FUNCTION_BLOCK FB_AdjustmentProcess
VAR_INPUT
    bEnable          : BOOL;
    bAbort           : BOOL;
    bStopRequest     : BOOL;
    bMachinePrepared : BOOL;
    bStartRequest    : BOOL;
    bDoneAck         : BOOL;

    // 与Screwdriver流程之间的保持型业务握手。
    bSecondTightenDone : BOOL;
    bReworkLoosenDone  : BOOL;

    // 保留原输入符号以兼容现有监控；协调器给它与二次拧紧Done相同的值。
    bRetractPermit : BOOL;
END_VAR

VAR_IN_OUT
    ioAdjustGripperAction : FB_GripperAction;
    ioAdjustGripper       : ST_GripperInterface;
    stAxisX               : ST_AxisInterface;
    stAxisY               : ST_AxisInterface;
    stAxisZ               : ST_AxisInterface;
END_VAR

VAR_OUTPUT
    bAdjustmentReady   : BOOL; // 兼容诊断：与二次拧紧请求保持一致
    bAdjustmentDone    : BOOL;
    bAdjustmentBusy    : BOOL;
    bAdjustmentQualified : BOOL;
	bAdjustmentOutOfRange : BOOL;
    bRequestSecondTighten : BOOL;
    bRequestReworkLoosen  : BOOL;// 当前件超出Adjustment可调整范围。
    bVisionTimeout     : BOOL;
    bVisionFault       : BOOL;
    bFallbackUsed      : BOOL;
    eVisionError       : E_VisionError := E_VisionError.None;
    fVisionCoaxiality  : LREAL;
    fCorrectionX       : LREAL;
    fCorrectionY       : LREAL;
    nAdjustCount       : UINT;
    nReworkCount       : UINT;
    bError             : BOOL;
    bGripperError      : BOOL;
    uiErrorAxis        : UINT;
    udErrorCode        : UDINT;
    eStep              : E_AdjustmentStep := E_AdjustmentStep.Idle;
    bAdjustGripperActionExecute : BOOL;
    eAdjustGripperActionCommand : E_GripperCommand := E_GripperCommand.None;
END_VAR

VAR
    fXWork : LREAL;
    fYWork : LREAL;
    fZWork : LREAL;
    fXStandby : LREAL;
    fYStandby : LREAL;
    fZSafe : LREAL;
    fXVelocity : LREAL;
    fYVelocity : LREAL;
    fZVelocity : LREAL;
    fPositionTolerance : LREAL;
    tMoveTimeout : TIME;

	//==============================================================
	// Adjustment最终被PLC接受并真正下发给轴的绝对目标
	//==============================================================
	fAdjustTargetX : LREAL;
	fAdjustTargetY : LREAL;
	
	
	//==============================================================
	// 本次Coax修正计算出的候选绝对目标
	//
	// Candidate = 当前实际位置 + Python修正量
	//
	// 候选值只有通过±最大修正范围检查后，
	// 才允许写入fAdjustTargetX/Y。
	//==============================================================
	fCandidateTargetX : LREAL;
	fCandidateTargetY : LREAL;
	
	
	//==============================================================
	// 修正目标范围诊断
	//==============================================================
	bCorrectionXOutOfRange : BOOL;
	bCorrectionYOutOfRange : BOOL;
	
	
	bVisionWithinTolerance : BOOL;
	
    fbMoveTimeout : TON;
    fbCoaxVision : FB_CoaxVision;
    // 当前逻辑检测点的额外检测计数；Retry路径不得清零。
    nCoaxRetryCount : UINT;
    fbCoaxRetryDelay : TON;
    bTimerRestart : BOOL;
    eTimedStep : E_AdjustmentStep := E_AdjustmentStep.Idle;
    bTimedMovement : BOOL;
    uiMovingAxis : UINT;

    bXIssued : BOOL;
    bYIssued : BOOL;
    bZIssued : BOOL;
    bXDone : BOOL;
    bYDone : BOOL;
    bZDone : BOOL;
END_VAR

// 沿用现有PositionConfig和MotionConfig；视觉工艺、次数和超时分别来自
// ProcessConfig与CommunicationConfig，FB内部不保存第二套参数源。
fXWork := GVL_PositionConfig.stAdjustment.stWork.X;
fYWork := GVL_PositionConfig.stAdjustment.stWork.Y;
fZWork := GVL_PositionConfig.stAdjustment.stWork.Z;
fXStandby := GVL_PositionConfig.stAdjustment.stReady.X;
fYStandby := GVL_PositionConfig.stAdjustment.stReady.Y;
fZSafe := GVL_PositionConfig.stAdjustment.stReady.Z;
fXVelocity := GVL_MotionConfig.stAdjustment.stX.fVelocity;
fYVelocity := GVL_MotionConfig.stAdjustment.stY.fVelocity;
fZVelocity := GVL_MotionConfig.stAdjustment.stZ.fVelocity;
fPositionTolerance := GVL_MotionConfig.stAdjustment.fPositionTolerance;
tMoveTimeout := GVL_MotionConfig.stAdjustment.tMoveTimeout;

bTimerRestart := (eStep <> eTimedStep);
eTimedStep := eStep;
bTimedMovement :=
    (eStep = E_AdjustmentStep.MoveXYToWork)
    OR (eStep = E_AdjustmentStep.LowerZToWork)
    OR (eStep = E_AdjustmentStep.WaitCorrectionXY)
    OR (eStep = E_AdjustmentStep.LiftZToSafe)
    OR (eStep = E_AdjustmentStep.ReturnXYToStandby);

IF bTimedMovement THEN
    CASE eStep OF
        E_AdjustmentStep.LowerZToWork,
        E_AdjustmentStep.LiftZToSafe:
            uiMovingAxis := GVL_AxisIndex.AdjustmentZ;

        E_AdjustmentStep.MoveXYToWork,
        E_AdjustmentStep.WaitCorrectionXY,
        E_AdjustmentStep.ReturnXYToStandby:
            IF NOT bXDone THEN
                uiMovingAxis := GVL_AxisIndex.AdjustmentX;
            ELSE
                uiMovingAxis := GVL_AxisIndex.AdjustmentY;
            END_IF;
    END_CASE;
END_IF;

fbMoveTimeout(
    IN := bEnable AND NOT bAbort AND bTimedMovement AND NOT bTimerRestart,
    PT := tMoveTimeout
);

stAxisX.AutoCmd.bMoveAbs := FALSE;
stAxisY.AutoCmd.bMoveAbs := FALSE;
stAxisZ.AutoCmd.bMoveAbs := FALSE;
bAdjustGripperActionExecute := FALSE;
eAdjustGripperActionCommand := E_GripperCommand.None;

// Retry属于Adjustment工艺层；两个Delay状态均撤销视觉bExecute。
// 每扫描只调用一次TON，离开Delay状态或停止/取消时复位。
fbCoaxRetryDelay(
    IN := bEnable AND NOT bAbort AND NOT bStopRequest
          AND ((eStep = E_AdjustmentStep.WaitMeasureRetryDelay)
               OR (eStep = E_AdjustmentStep.WaitFinalMeasureRetryDelay)),
    PT := GVL_ProcessConfig.stAdjustment.tCoaxRetryDelay
);

// Process只保持执行请求并消费强类型结果；ADS、RequestId、ResultId和Timeout
// 全部封装在FB_CoaxVision -> FB_VisionRequest中。
fbCoaxVision(
    bExecute := bEnable
                AND NOT bAbort
                AND
                (
                    (eStep = E_AdjustmentStep.WaitMeasureResult)
                    OR (eStep = E_AdjustmentStep.WaitFinalMeasure)
                ),
    bCancel := bStopRequest OR bAbort
);

IF NOT bEnable OR bAbort THEN
    IF bMachinePrepared THEN
        ioAdjustGripperAction(
            bExecute := FALSE,
            eCommand := E_GripperCommand.None,
            bCancel := bStopRequest OR bAbort,
            tAcceptTimeout := GVL_ProcessConfig.stGripper.tAcceptTimeout,
            tResultTimeout := GVL_ProcessConfig.stGripper.tResultTimeout,
            ioGripper := ioAdjustGripper
        );
    END_IF;

    bAdjustmentReady := FALSE;
    bAdjustmentDone := FALSE;
    bAdjustmentBusy := FALSE;
    bAdjustmentQualified := FALSE;
	bAdjustmentOutOfRange := FALSE;
    bRequestSecondTighten := FALSE;
    bRequestReworkLoosen := FALSE;
    bVisionTimeout := FALSE;
    bVisionFault := FALSE;
    bFallbackUsed := FALSE;
    eVisionError := E_VisionError.None;
    fCorrectionX := 0.0;
    fCorrectionY := 0.0;
	fCandidateTargetX := 0.0;
	fCandidateTargetY := 0.0;
	bCorrectionXOutOfRange := FALSE;
	bCorrectionYOutOfRange := FALSE;
    nAdjustCount := 0;
    nReworkCount := 0;
    nCoaxRetryCount := 0;
    bError := FALSE;
    bGripperError := FALSE;
    uiErrorAxis := 0;
    udErrorCode := TO_UDINT(E_ScrewdriverErrorCode.None);
    bXIssued := FALSE;
    bYIssued := FALSE;
    bZIssued := FALSE;
    bXDone := FALSE;
    bYDone := FALSE;
    bZDone := FALSE;
    eStep := E_AdjustmentStep.Idle;
    RETURN;
END_IF;

IF (eStep = E_AdjustmentStep.Idle) AND bStartRequest THEN

 	//==========================================================
    // 新工件开始，清除上一件质量结果。
    //==========================================================
    bAdjustmentQualified := FALSE;
	bAdjustmentOutOfRange := FALSE;

    bVisionTimeout := FALSE;
    bVisionFault := FALSE;
    bFallbackUsed := FALSE;
    eVisionError := E_VisionError.None;

    bVisionWithinTolerance := FALSE;

    fVisionCoaxiality := 0.0;

    fCorrectionX := 0.0;
    fCorrectionY := 0.0;

    // 初始接受目标仍然从Adjustment工作位置开始。
    fAdjustTargetX := fXWork;
    fAdjustTargetY := fYWork;

    // 候选目标初始化到工作位置。
    fCandidateTargetX := fXWork;
    fCandidateTargetY := fYWork;

    // 清除上一件产品的范围诊断。
    bCorrectionXOutOfRange := FALSE;
    bCorrectionYOutOfRange := FALSE;

    nAdjustCount := 0;
    nReworkCount := 0;
    nCoaxRetryCount := 0;

    bXIssued := FALSE;
    bYIssued := FALSE;
    bXDone := FALSE;
    bYDone := FALSE;

    eStep := E_AdjustmentStep.MoveXYToWork;
END_IF;

// 准备阶段结束后，COM4命令权归本FB；Open持续到最终质量结果确定。
IF bMachinePrepared THEN
    IF eStep = E_AdjustmentStep.OpenGripper THEN
        bAdjustGripperActionExecute := TRUE;
        eAdjustGripperActionCommand := E_GripperCommand.Open;
    ELSIF eStep = E_AdjustmentStep.CloseGripper THEN
        bAdjustGripperActionExecute := TRUE;
        eAdjustGripperActionCommand := E_GripperCommand.Close;
    END_IF;

    ioAdjustGripperAction(
        bExecute := bAdjustGripperActionExecute,
        eCommand := eAdjustGripperActionCommand,
        bCancel := bStopRequest OR bAbort,
        tAcceptTimeout := GVL_ProcessConfig.stGripper.tAcceptTimeout,
        tResultTimeout := GVL_ProcessConfig.stGripper.tResultTimeout,
        ioGripper := ioAdjustGripper
    );
END_IF;

IF stAxisX.Alarm.bError OR stAxisY.Alarm.bError OR stAxisZ.Alarm.bError THEN
    bError := TRUE;
    bGripperError := FALSE;
    eStep := E_AdjustmentStep.Error;
    IF stAxisX.Alarm.bError THEN
        uiErrorAxis := GVL_AxisIndex.AdjustmentX;
        udErrorCode := stAxisX.Alarm.nErrorID;
    ELSIF stAxisY.Alarm.bError THEN
        uiErrorAxis := GVL_AxisIndex.AdjustmentY;
        udErrorCode := stAxisY.Alarm.nErrorID;
    ELSE
        uiErrorAxis := GVL_AxisIndex.AdjustmentZ;
        udErrorCode := stAxisZ.Alarm.nErrorID;
    END_IF;
END_IF;

IF ioAdjustGripperAction.bError
    AND ((eStep = E_AdjustmentStep.OpenGripper)
         OR (eStep = E_AdjustmentStep.CloseGripper))
THEN
    bError := TRUE;
    bGripperError := TRUE;
    uiErrorAxis := 0;
    IF ioAdjustGripperAction.udErrorCode <> 0 THEN
        udErrorCode := ioAdjustGripperAction.udErrorCode;
    ELSE
        udErrorCode := TO_UDINT(E_ScrewdriverErrorCode.AdjustmentGripperFailed);
    END_IF;
    eStep := E_AdjustmentStep.Error;
END_IF;

IF fbMoveTimeout.Q AND NOT bError THEN
    bError := TRUE;
    bGripperError := FALSE;
    uiErrorAxis := uiMovingAxis;
    udErrorCode := TO_UDINT(E_ScrewdriverErrorCode.PositionTimeout);
    eStep := E_AdjustmentStep.Error;
END_IF;

CASE eStep OF
    E_AdjustmentStep.Idle:
        bAdjustmentDone := FALSE;

    E_AdjustmentStep.MoveXYToWork:
        IF NOT bXDone THEN
            bXDone := M_MoveAxisAbsolute(fTarget := fXWork, fVelocity := fXVelocity,
                uiAxis := GVL_AxisIndex.AdjustmentX, ioIssued := bXIssued, ioAxis := stAxisX);
        END_IF;
        IF NOT bYDone THEN
            bYDone := M_MoveAxisAbsolute(fTarget := fYWork, fVelocity := fYVelocity,
                uiAxis := GVL_AxisIndex.AdjustmentY, ioIssued := bYIssued, ioAxis := stAxisY);
        END_IF;
        IF bXDone AND bYDone THEN
            fAdjustTargetX := fXWork;
            fAdjustTargetY := fYWork;
            bZIssued := FALSE;
            bZDone := FALSE;
            eStep := E_AdjustmentStep.LowerZToWork;
        END_IF;

    E_AdjustmentStep.LowerZToWork:
        bZDone := M_MoveAxisAbsolute(fTarget := fZWork, fVelocity := fZVelocity,
            uiAxis := GVL_AxisIndex.AdjustmentZ, ioIssued := bZIssued, ioAxis := stAxisZ);
        IF bZDone THEN
            eStep := E_AdjustmentStep.OpenGripper;
        END_IF;

    E_AdjustmentStep.OpenGripper:
        IF ioAdjustGripperAction.bDone THEN
            eStep := E_AdjustmentStep.PrepareMeasurement;
        END_IF;

    E_AdjustmentStep.PrepareMeasurement:
        // 工作位的首次逻辑检测点。Retry直接回RequestMeasure，不经过这里。
        nCoaxRetryCount := 0;
        fCorrectionX := 0.0;
        fCorrectionY := 0.0;
        bVisionWithinTolerance := FALSE;
        // Simulation与Camera都从FB_CoaxVision的统一结果出口获取数据。
        eStep := E_AdjustmentStep.RequestMeasure;

    E_AdjustmentStep.RequestMeasure:
        fCorrectionX := 0.0;
        fCorrectionY := 0.0;
        bVisionWithinTolerance := FALSE;
        eStep := E_AdjustmentStep.WaitMeasureResult;

    E_AdjustmentStep.WaitMeasureResult:
        // Cancelled/Stop由现有Stop/Abort/Reset体系清理，不消费为产品结果。
        IF fbCoaxVision.bDone
            AND NOT bStopRequest
            AND (fbCoaxVision.eVisionError <> E_VisionError.Cancelled)
        THEN
            IF fbCoaxVision.bVisionFault THEN
                IF ((fbCoaxVision.eVisionError = E_VisionError.InvalidResult)
                    OR (fbCoaxVision.eVisionError = E_VisionError.Timeout))
                    AND (nCoaxRetryCount < GVL_ProcessConfig.stAdjustment.nCoaxMaxRetryCount)
                THEN
                    // 暂时失败不锁存工件级诊断；下一次执行创建新的RequestId。
                    nCoaxRetryCount := nCoaxRetryCount + 1;
                    eStep := E_AdjustmentStep.WaitMeasureRetryDelay;
                ELSE
                    // Retry耗尽，或Offline/ServiceFault：当前件不合格，正常撤离。
                    bVisionFault := TRUE;
                    bFallbackUsed := fbCoaxVision.bFallbackUsed;
                    eVisionError := fbCoaxVision.eVisionError;
                    bVisionTimeout :=
                        fbCoaxVision.eVisionError = E_VisionError.Timeout;
                    bAdjustmentQualified := FALSE;
                    eStep := E_AdjustmentStep.CloseGripper;
                END_IF;
            ELSE
                // 仅有效测量进入工艺判断；恢复成功不保留中间失败诊断。
                bVisionFault := FALSE;
                bVisionTimeout := FALSE;
                bFallbackUsed := FALSE;
                eVisionError := E_VisionError.None;
                fVisionCoaxiality := fbCoaxVision.stResult.fCoaxiality;
                fCorrectionX := fbCoaxVision.stResult.fCorrectionX;
                fCorrectionY := fbCoaxVision.stResult.fCorrectionY;
                bVisionWithinTolerance :=
                    fVisionCoaxiality <= GVL_ProcessConfig.stAdjustment.fAdjustTolerance;
                eStep := E_AdjustmentStep.EvaluateAdjustment;
            END_IF;
        END_IF;

    E_AdjustmentStep.WaitMeasureRetryDelay:
        // 本扫描fbCoaxVision.bExecute=FALSE，PT=0时也先正常复位旧事务。
        IF fbCoaxRetryDelay.Q AND NOT bStopRequest THEN
            // 同一逻辑检测点的Retry，保留nCoaxRetryCount。
            eStep := E_AdjustmentStep.RequestMeasure;
        END_IF;

    E_AdjustmentStep.EvaluateAdjustment:

		//==========================================================
		// 情况1：
		// 当前同轴度已经达到调整容差；
		//
		// 或者：
		// 已经达到本轮最大允许调整次数。
		//
		// 此时不再进行新的AdjustmentXY修正。
		//==========================================================
		IF
			bVisionWithinTolerance
			OR
			(
				nAdjustCount
				>= GVL_ProcessConfig.stAdjustment.nMaxAdjustCount
			)
		THEN
	
			eStep :=
				E_AdjustmentStep.RequestSecondTighten;
	
	
		ELSE
	
			//======================================================
			// 统一视觉结果中的Correction为机械相对修正位移，单位mm。
			// Camera映射与比例标定由Python完成；Simulation由FB_CoaxVision生成。
			// 本流程直接消费Correction，不再根据Delta映射或换算。
			// Candidate = ActualPosition + Correction
			//======================================================	
			fCandidateTargetX :=
				stAxisX.Data.fActPosition
				+ fCorrectionX;
	
			fCandidateTargetY :=
				stAxisY.Data.fActPosition
				+ fCorrectionY;
	
	
			//======================================================
			// 检查候选位置是否仍然处于
			//
			// Adjustment工作位置 ± 最大允许调整范围
			//
			// 这里检查的是累计机械偏移，
			// 而不是单次Delta大小。
			//======================================================
	
			bCorrectionXOutOfRange :=
				ABS(
					fCandidateTargetX
					- fXWork
				)
				>
				GVL_ProcessConfig.stAdjustment.fMaxCorrectionX;
	
			bCorrectionYOutOfRange :=
				ABS(
					fCandidateTargetY
					- fYWork
				)
				>
				GVL_ProcessConfig.stAdjustment.fMaxCorrectionY;
	
	
			//======================================================
			// 任意一个方向越界：
			//
			// X/Y作为同一次二维Coax修正，
			// 不允许只执行其中一根轴。
			//
			// 所以两根轴都不运动。
			//======================================================
			IF
				bCorrectionXOutOfRange
				OR
				bCorrectionYOutOfRange
			THEN
			
				// 超范围仅是调整能力诊断；不接受Candidate，不移动任意一根轴。
				// 仍执行二次拧紧，最终质量仅由Final Coax决定。
				bAdjustmentOutOfRange := TRUE;
				bXIssued := FALSE;
				bYIssued := FALSE;
				bXDone := FALSE;
				bYDone := FALSE;
				eStep := E_AdjustmentStep.RequestSecondTighten;

			ELSE
			
				//==========================================================
				// X/Y候选目标均处于允许Adjustment修正窗口内。
				// 正式接受Candidate作为新的轴绝对目标。
				//==========================================================
			
				bAdjustmentOutOfRange := FALSE;
			
				fAdjustTargetX :=
					fCandidateTargetX;
			
				fAdjustTargetY :=
					fCandidateTargetY;
			
				nAdjustCount :=
					nAdjustCount + 1;
			
				eStep :=
					E_AdjustmentStep.StartCorrectionXY;
			
			END_IF;

		END_IF;

    E_AdjustmentStep.StartCorrectionXY:
        bXIssued := FALSE;
        bYIssued := FALSE;
        bXDone := FALSE;
        bYDone := FALSE;
        eStep := E_AdjustmentStep.WaitCorrectionXY;

    E_AdjustmentStep.WaitCorrectionXY:
        // Z保持工作高度，X/Y同时向通过工艺范围检查后的绝对目标运动。
        IF NOT bXDone THEN
            bXDone := M_MoveAxisAbsolute(fTarget := fAdjustTargetX, fVelocity := fXVelocity,
                uiAxis := GVL_AxisIndex.AdjustmentX, ioIssued := bXIssued, ioAxis := stAxisX);
        END_IF;
        IF NOT bYDone THEN
            bYDone := M_MoveAxisAbsolute(fTarget := fAdjustTargetY, fVelocity := fYVelocity,
                uiAxis := GVL_AxisIndex.AdjustmentY, ioIssued := bYIssued, ioAxis := stAxisY);
        END_IF;
        IF bXDone AND bYDone THEN
            // 每次XY修正完成后开始新的逻辑检测点。
            nCoaxRetryCount := 0;
            eStep := E_AdjustmentStep.RequestMeasure;
        END_IF;

    E_AdjustmentStep.RequestSecondTighten:
        eStep := E_AdjustmentStep.WaitSecondTighten;

    E_AdjustmentStep.WaitSecondTighten:
        IF bSecondTightenDone OR bRetractPermit THEN
            // 二次拧紧已完成；Final是独立的逻辑检测点。
            nCoaxRetryCount := 0;
            eStep := E_AdjustmentStep.RequestFinalMeasure;
        END_IF;

    E_AdjustmentStep.RequestFinalMeasure:
        fCorrectionX := 0.0;
        fCorrectionY := 0.0;
        bVisionWithinTolerance := FALSE;
        eStep := E_AdjustmentStep.WaitFinalMeasure;

    E_AdjustmentStep.WaitFinalMeasure:
        // Cancelled/Stop由现有Stop/Abort/Reset体系清理，不消费为产品结果。
        IF fbCoaxVision.bDone
            AND NOT bStopRequest
            AND (fbCoaxVision.eVisionError <> E_VisionError.Cancelled)
        THEN
            IF fbCoaxVision.bVisionFault THEN
                IF ((fbCoaxVision.eVisionError = E_VisionError.InvalidResult)
                    OR (fbCoaxVision.eVisionError = E_VisionError.Timeout))
                    AND (nCoaxRetryCount < GVL_ProcessConfig.stAdjustment.nCoaxMaxRetryCount)
                THEN
                    // 暂时失败不锁存工件级诊断；下一次执行创建新的RequestId。
                    nCoaxRetryCount := nCoaxRetryCount + 1;
                    eStep := E_AdjustmentStep.WaitFinalMeasureRetryDelay;
                ELSE
                    // Retry耗尽，或Offline/ServiceFault：当前件不合格，正常撤离。
                    bVisionFault := TRUE;
                    bFallbackUsed := fbCoaxVision.bFallbackUsed;
                    eVisionError := fbCoaxVision.eVisionError;
                    bVisionTimeout :=
                        fbCoaxVision.eVisionError = E_VisionError.Timeout;
                    bAdjustmentQualified := FALSE;
                    eStep := E_AdjustmentStep.CloseGripper;
                END_IF;
            ELSE
                // 仅有效测量进入工艺判断；恢复成功不保留中间失败诊断。
                bVisionFault := FALSE;
                bVisionTimeout := FALSE;
                bFallbackUsed := FALSE;
                eVisionError := E_VisionError.None;
                fVisionCoaxiality := fbCoaxVision.stResult.fCoaxiality;
                fCorrectionX := fbCoaxVision.stResult.fCorrectionX;
                fCorrectionY := fbCoaxVision.stResult.fCorrectionY;
                bVisionWithinTolerance :=
                    fVisionCoaxiality <= GVL_ProcessConfig.stAdjustment.fQualifiedTolerance;
                eStep := E_AdjustmentStep.EvaluateFinalResult;
            END_IF;
        END_IF;

    E_AdjustmentStep.WaitFinalMeasureRetryDelay:
        // 本扫描fbCoaxVision.bExecute=FALSE，PT=0时也先正常复位旧事务。
        IF fbCoaxRetryDelay.Q AND NOT bStopRequest THEN
            // 同一逻辑检测点的Retry，保留nCoaxRetryCount。
            eStep := E_AdjustmentStep.RequestFinalMeasure;
        END_IF;

    E_AdjustmentStep.EvaluateFinalResult:
        IF bVisionWithinTolerance THEN
            // Final有效且合格：不返工。
            bAdjustmentQualified := TRUE;
            eStep := E_AdjustmentStep.CloseGripper;

        ELSIF nReworkCount < GVL_ProcessConfig.stAdjustment.nMaxReworkCount THEN
            // Final有效超差且仍有返工额度：只计数一次，进入既有拧松状态。
            nReworkCount := nReworkCount + 1;
            bAdjustmentQualified := FALSE;
            eStep := E_AdjustmentStep.RequestReworkLoosen;

        ELSE
            // Final有效超差且额度耗尽：NG并正常撤离。
            bAdjustmentQualified := FALSE;
            eStep := E_AdjustmentStep.CloseGripper;
        END_IF;

    // 复用既有返工拧松握手；完成后直接返回原检测调整循环。
    E_AdjustmentStep.RequestReworkLoosen:
        eStep := E_AdjustmentStep.WaitReworkLoosen;

    E_AdjustmentStep.WaitReworkLoosen:
        IF bReworkLoosenDone THEN
            // AdjustmentXYZ与COM4始终未撤离；仅重置本轮修正和视觉重试计数并重新检测。
            nAdjustCount := 0;
            nCoaxRetryCount := 0;
            fCorrectionX := 0.0;
            fCorrectionY := 0.0;
            bVisionWithinTolerance := FALSE;
            eStep := E_AdjustmentStep.RequestMeasure;
        END_IF;

    E_AdjustmentStep.CloseGripper:
        IF ioAdjustGripperAction.bDone THEN
            bZIssued := FALSE;
            bZDone := FALSE;
            eStep := E_AdjustmentStep.LiftZToSafe;
        END_IF;

    E_AdjustmentStep.LiftZToSafe:
        bZDone := M_MoveAxisAbsolute(fTarget := fZSafe, fVelocity := fZVelocity,
            uiAxis := GVL_AxisIndex.AdjustmentZ, ioIssued := bZIssued, ioAxis := stAxisZ);
        IF bZDone THEN
            bXIssued := FALSE;
            bYIssued := FALSE;
            bXDone := FALSE;
            bYDone := FALSE;
            eStep := E_AdjustmentStep.ReturnXYToStandby;
        END_IF;

    E_AdjustmentStep.ReturnXYToStandby:
        IF NOT bXDone THEN
            bXDone := M_MoveAxisAbsolute(fTarget := fXStandby, fVelocity := fXVelocity,
                uiAxis := GVL_AxisIndex.AdjustmentX, ioIssued := bXIssued, ioAxis := stAxisX);
        END_IF;
        IF NOT bYDone THEN
            bYDone := M_MoveAxisAbsolute(fTarget := fYStandby, fVelocity := fYVelocity,
                uiAxis := GVL_AxisIndex.AdjustmentY, ioIssued := bYIssued, ioAxis := stAxisY);
        END_IF;
        IF bXDone AND bYDone THEN
            bAdjustmentDone := TRUE;
            eStep := E_AdjustmentStep.WaitDoneAck;
        END_IF;

    E_AdjustmentStep.WaitDoneAck:
        bAdjustmentDone := TRUE;
        IF bDoneAck THEN
            nCoaxRetryCount := 0;
            bAdjustmentDone := FALSE;
            bAdjustmentQualified := FALSE;
            bXIssued := FALSE;
            bYIssued := FALSE;
            bZIssued := FALSE;
            bXDone := FALSE;
            bYDone := FALSE;
            bZDone := FALSE;
            eStep := E_AdjustmentStep.Idle;
        END_IF;

    E_AdjustmentStep.Error:
        bAdjustmentDone := FALSE;
        bError := TRUE;
END_CASE;

// 保持型握手由状态直接派生，避免单扫描脉冲丢失。
bRequestSecondTighten :=
    (eStep = E_AdjustmentStep.RequestSecondTighten)
    OR (eStep = E_AdjustmentStep.WaitSecondTighten);
bAdjustmentReady := bRequestSecondTighten;
bRequestReworkLoosen :=
    (eStep = E_AdjustmentStep.RequestReworkLoosen)
    OR (eStep = E_AdjustmentStep.WaitReworkLoosen);

IF eStep = E_AdjustmentStep.OpenGripper THEN
    bAdjustGripperActionExecute := TRUE;
    eAdjustGripperActionCommand := E_GripperCommand.Open;
ELSIF eStep = E_AdjustmentStep.CloseGripper THEN
    bAdjustGripperActionExecute := TRUE;
    eAdjustGripperActionCommand := E_GripperCommand.Close;
ELSE
    bAdjustGripperActionExecute := FALSE;
    eAdjustGripperActionCommand := E_GripperCommand.None;
END_IF;

bAdjustmentBusy :=
    (eStep <> E_AdjustmentStep.Idle)
    AND (eStep <> E_AdjustmentStep.Error);

METHOD PRIVATE M_MoveAxisAbsolute : BOOL
VAR_INPUT
    fTarget   : LREAL;
    fVelocity : LREAL;
    uiAxis    : UINT;
END_VAR
VAR_IN_OUT
    ioIssued : BOOL;
    ioAxis   : ST_AxisInterface;
END_VAR
M_MoveAxisAbsolute := FALSE;

IF ioAxis.Alarm.bError THEN
    ioIssued := FALSE;
    RETURN;
END_IF;

IF ioAxis.State.bReady
    AND NOT ioAxis.State.bBusy
    AND NOT ioAxis.State.bActive
    AND (ABS(ioAxis.Data.fActPosition - fTarget) <= fPositionTolerance)
THEN
    ioIssued := FALSE;
    M_MoveAxisAbsolute := TRUE;
    RETURN;
END_IF;

IF NOT ioIssued THEN
    IF NOT ioAxis.State.bReady OR ioAxis.State.bBusy OR ioAxis.State.bActive THEN
        RETURN;
    END_IF;

    ioAxis.AutoSet.Position.fAbsolutePosition := fTarget;
    ioAxis.AutoSet.Position.fVelocity := fVelocity;
    ioAxis.AutoCmd.bMoveAbs := TRUE;
    ioIssued := TRUE;
    RETURN;
END_IF;

IF ioAxis.State.bCmdRejected OR ioAxis.State.bCommandAborted THEN
    bError := TRUE;
    bGripperError := FALSE;
    uiErrorAxis := uiAxis;
    udErrorCode := TO_UDINT(E_ScrewdriverErrorCode.AdjustmentCommandFailed);
    ioIssued := FALSE;
    eStep := E_AdjustmentStep.Error;
    RETURN;
END_IF;

IF ioAxis.State.bReady
    AND NOT ioAxis.State.bBusy
    AND (ABS(ioAxis.Data.fActPosition - fTarget) <= fPositionTolerance)
THEN
    ioIssued := FALSE;
    M_MoveAxisAbsolute := TRUE;
END_IF;
END_METHOD

END_FUNCTION_BLOCK

(* stored: Version 1.1.0.1, ProductVersion 3.1.4026.20
   POU FB_AdjustmentProcess: Id {6be3f419-7e42-4f1c-ad50-7db14f957959}, SpecialFunc None
   Method M_MoveAxisAbsolute: Id {d92a53a5-1112-4138-b128-19cd21bfd66f} *)
